(*
SPDX-FileCopyrightText: © 2026 Oleksandr Tiutyk <trofimich@gmail.com>
SPDX-License-Identifier: MIT
License: https://opensource.org/license/mit
*)

(*!
<summary>Provides byte sequence mutation and raw-memory copying.</summary>
<description>
Append adds bytes. LoadFrom writes at startIndex and sets Length to the end of the copied range, potentially
truncating the old tail. Input memory is borrowed for copying, never adopted. Remove by value is a no-op when
the value is absent, including on an empty collection. See method declarations for current safety limitations.
</description>
*)

INTERFACE IByteList EXTENDS IReadOnlyByteList

(*!
<summary>Appends the raw storage bytes of an ANY argument.</summary>
<description>
Borrows the argument for copying and uses its full runtime size, including string capacity and structure
padding. Not portable serialization or object cloning. Shares AppendData capacity checks, overlap support and
failure behavior.
</description>
*)
METHOD AppendAny : IByteList
VAR_INPUT
	data : ANY;
END_VAR
END_METHOD

(*!
<summary>Appends one byte by value.</summary>
<description>
Returns this list. Full static storage raises an exception; dynamic growth uses checked allocation and
terminal OOM handling.
</description>
*)
METHOD AppendByte : IByteList
VAR_INPUT
	value : BYTE;
END_VAR
END_METHOD

(*!
<summary>Appends bytes copied from a borrowed memory range.</summary>
<description>
Null data or zero dataSize is a no-op before size validation. Otherwise the source must be readable and
negative sizes or a resulting length outside DINT raise ArgumentOutOfRangeException before copying. Static
capacity exhaustion raises StaticCollectionFullException. Dynamic allocation uses checked growth and terminal
OOM handling. The existing growth increment (free capacity plus input size) is retained and must also fit. The
source may refer to this collection buffer, including overlapping ranges. The caller must provide a readable
range of dataSize bytes; growth keeps the old buffer alive until copying completes. No restriction to logical
Length is imposed on the source. Returns this list.
</description>
*)
METHOD AppendData : IByteList
VAR_INPUT
	data : POINTER TO BYTE;
	dataSize : TOF_Core.DINT_LENGTH;
END_VAR
END_METHOD

(*!
<summary>Appends the raw bytes referenced by a generic descriptor.</summary>
<description>
Borrows the descriptor without adopting or releasing it. Copies Address and Size without value conversion or
object cloning. Size above SignedInt32.MAX_VALUE raises ArgumentOutOfRangeException before narrowing,
including for a null Address. Shares AppendData aliasing and failure behavior.
</description>
*)
METHOD AppendGeneric : IByteList
VAR_INPUT
	data : TOF_Core.GENERIC_VALUE;
END_VAR
END_METHOD

(*!
<summary>Resets the byte count and optionally releases dynamic storage.</summary>
<description>
The default retains capacity for reuse. releaseDynamicMemory = TRUE deletes dynamic storage and sets capacity
to zero. Static storage is retained. Returns this list; old contents are no longer logical entries.
</description>
*)
METHOD Clear : IByteList
VAR_INPUT
	releaseDynamicMemory : BOOL := FALSE;
END_VAR
END_METHOD

(*!
<summary>Loads the full raw representation of an ANY argument at a position.</summary>
<description>
Delegates to LoadFromData using the runtime byte size, including padding and string capacity. Borrows the
source and may truncate the previous tail. Shares LoadFromData limits; not portable serialization.
</description>
*)
METHOD LoadFromAny : IByteList
VAR_INPUT
	data : ANY;
	startIndex : TOF_Core.DINT_INDEX := 0;
END_VAR
END_METHOD

(*!
<summary>Copies bytes at a position and sets Length to the end of the copy.</summary>
<description>
startIndex must lie between zero and old Length inclusive, and dataSize must be nonnegative; invalid arguments
raise ArgumentOutOfRangeException. Null data or zero size leaves Length unchanged after these checks. For a
nonempty copy, the resulting length is checked against DINT before arithmetic or mutation. The prefix remains
and the tail beyond the new end is logically truncated. Static capacity exhaustion raises
StaticCollectionFullException; dynamic growth uses checked allocation and terminal OOM handling. Internal
sources and overlapping ranges are supported. The caller must provide a readable source range of dataSize
bytes; the old buffer remains alive throughout copying on growth. No restriction to logical Length is imposed
on the source. Returns this list.
</description>
*)
METHOD LoadFromData : IByteList
VAR_INPUT
	data : POINTER TO BYTE;
	dataSize : TOF_Core.DINT_LENGTH;
	startIndex : TOF_Core.DINT_INDEX := 0;
END_VAR
END_METHOD

(*!
<summary>Loads the byte range referenced by a generic descriptor.</summary>
<description>
Borrows the descriptor without adoption or release. Size above SignedInt32.MAX_VALUE raises
ArgumentOutOfRangeException before narrowing, including for a null Address. Shares LoadFromData index checks,
truncation, aliasing and failure behavior.
</description>
*)
METHOD LoadFromGeneric : IByteList
VAR_INPUT
	data : TOF_Core.GENERIC_VALUE;
	startIndex : TOF_Core.DINT_INDEX := 0;
END_VAR
END_METHOD

(*!
<summary>Removes the first occurrence of a byte if present.</summary>
<description>
Removes only the first matching byte, compacts later bytes through RemoveAt and returns this list. An absent
value or an empty static or dynamic list leaves the collection unchanged without raising an exception for
absence. Capacity is retained. Requires an intact collection whose backing storage remains valid for its
logical contents.
</description>
*)
METHOD Remove : IByteList
VAR_INPUT
	value : BYTE;
END_VAR
END_METHOD

(*!
<summary>Removes a contiguous byte range and compacts remaining bytes.</summary>
<description>
Requires an existing index and a nonnegative count no greater than the remaining length; otherwise raises
ArgumentOutOfRangeException. The range is checked by subtraction before computing its end. Zero count is a
no-op only after index validation. Capacity is retained. Returns this list.
</description>
*)
METHOD RemoveAt : IByteList
VAR_INPUT
	index : TOF_Core.DINT_INDEX;
	count : TOF_Core.DINT_LENGTH := 1;
END_VAR
END_METHOD

(*!
<summary>Overwrites one existing byte.</summary>
<description>
Requires allocated storage and an index within Length; otherwise raises an exception. Length and Capacity are
unchanged. Returns this list.
</description>
*)
METHOD Set : IByteList
VAR_INPUT
	index : TOF_Core.DINT_INDEX;
	value : BYTE;
END_VAR
END_METHOD

END_INTERFACE

(* stored: Version 1.1.0.1
   Itf IByteList: Id {518eb55c-df07-0206-0227-e692a273d945}
   Method AppendAny: Id {1b640082-c494-4770-8a43-3eb7addbc09e}
   Method AppendByte: Id {1ab7d3cb-0dd2-4a95-871a-2df749dcb5a5}
   Method AppendData: Id {1186b88b-e5f6-4d0a-850c-7b49aca8e28d}
   Method AppendGeneric: Id {c20b42af-40c5-495e-b096-4ffb90d5ad93}
   Method Clear: Id {243fdc07-7928-4ca7-a298-f89f02bbd736}
   Method LoadFromAny: Id {b3c42220-f6d9-4c15-b9b4-e89b6fac55f8}
   Method LoadFromData: Id {f1c6da5c-ced0-42ee-9f57-c45302a7ebcb}
   Method LoadFromGeneric: Id {0e129b3d-d8f7-4a58-8e16-3c8b5d4146dc}
   Method Remove: Id {eed9e02a-e972-481f-8ddf-d0d8fccc576a}
   Method RemoveAt: Id {5d545c6c-7499-43af-8e59-315db670ead5}
   Method Set: Id {267c54d8-2df6-0ce5-162c-03537dc39a04} *)
